PROGRAM VisuLogic
VAR_OUTPUT
	L_Run: BOOL;
	L_StopOP: BOOL;
	L_StopEM: BOOL;
	L_Manual: BOOL;
	
	
END_VAR
VAR
	T_StopOP: TON;
	Time_Stop: TIME := T#1S;
END_VAR


L_Run := (GVL.Mode = Modes.AUTO);
L_Manual := (GVL.Mode = Modes.MAN);
L_StopEM := (GVL.Mode = Modes.STOP_EM);
IF GVL.Mode <> Modes.STOP_OP THEN
	L_stopOP := FALSE;
END_IF

//Timing Stop OP
IF GVL.Mode = Modes.STOP_OP THEN
	T_StopOP(IN:=TRUE, PT:=Time_Stop);
	IF T_StopOP.Q THEN
		T_StopOP(IN:=FALSE);
		L_StopOP := NOT L_StopOP;
	END_IF
END_IF

END_PROGRAM

(* stored: Version 1.1.0.1, ProductVersion 3.1.4024.9
   POU VisuLogic: Id {8922458d-0421-4f98-b48e-184c3c0cea3c}, SpecialFunc None *)
